# EPICS autosave request: TimRxApp/Db/TimRx_settings.req
file "TimRxCfg_settings.req",         P=$(P), R=$(R)
file "TimRxAMCTrigCh_settings.req",   P=$(P), R=$(R)
file "TimRxFMCTrigCh_settings.req",   P=$(P), R=$(R)
